// TIA Portal V17 export
// export: Created 2024-08-29T18:23:43.9946444Z, ExportSetting WithDefaults, DisplayName Totally Integrated Automation Portal, DisplayVersion V17 Update 7, DisplayName TIA Portal Openness, DisplayVersion V17 Update 7, DisplayName TIA Portal Version Control Interface, DisplayVersion V17, DisplayName SINAMICS Startdrive Advanced, DisplayVersion V17 SP2, DisplayName SINAMICS Startdrive G110M, G120, G120C, G120D, G120P, G115D, DisplayVersion V17 SP2, DisplayName SINAMICS Startdrive G130, G150, S120, S150, SINAMICS MV, S210, DisplayVersion V17 SP2, DisplayName STEP 7 Professional, DisplayVersion V17 Update 7, DisplayName STEP 7 Safety, DisplayVersion V17 Update 6, DisplayName WinCC Advanced / Unified PC, DisplayVersion V17 Update 7
DATA_BLOCK "motor"   // DB19
{ S7_Optimized_Access := 'TRUE' }
VERSION : 0.1
// stored: AutoNumber true, DBAccessibleFromOPCUA true, DBAccessibleFromWebserver true, IsOnlyStoredInLoadMemory false, IsRetainMemResEnabled false, IsWriteProtectedInAS false, MemoryReserve 100
   VAR RETAIN
      on : Bool := TRUE;
      track1Test : Bool := FALSE;
      track2Test : Bool := FALSE;
      pulseNumber1 : Int := 5;
      waitTime1 : DInt := 100;
      pulseWidth2 : DInt := 10;
      cicleTime2 : DInt := 200;
      pulseNumber2 : Int := 5;
      waitTime2 : DInt := 100;
      cicleTime1 : DInt := 200;
      pulseWidth1 : DInt := 10;
   END_VAR
BEGIN
END_DATA_BLOCK
